{attribute addProperty BoxType "EL6201-0000-0017"}
{attribute addProperty Id "Slave_28A_DI0BIT10.125217Slave_28A_DI1BIT10.125218Slave_28A_DI2BIT10.125219Slave_28A_DI3BIT10.125220Slave_28B_DI0BIT10.125221Slave_28B_DI1BIT10.125222Slave_28B_DI2BIT10.125223Slave_28B_DI3BIT10.125224"}
{attribute addProperty CRC "1401413082"}
{attribute addProperty SizeInBites "8"}
{attribute addProperty SizeInBytes "1"}
TYPE Slave_28_Inputs_5387DDDA :
STRUCT
	{attribute addProperty Name "Slave_28A_DI0"}
	Slave_28A_DI0 : BIT;
	{attribute addProperty Name "Slave_28A_DI1"}
	Slave_28A_DI1 : BIT;
	{attribute addProperty Name "Slave_28A_DI2"}
	Slave_28A_DI2 : BIT;
	{attribute addProperty Name "Slave_28A_DI3"}
	Slave_28A_DI3 : BIT;
	{attribute addProperty Name "Slave_28B_DI0"}
	Slave_28B_DI0 : BIT;
	{attribute addProperty Name "Slave_28B_DI1"}
	Slave_28B_DI1 : BIT;
	{attribute addProperty Name "Slave_28B_DI2"}
	Slave_28B_DI2 : BIT;
	{attribute addProperty Name "Slave_28B_DI3"}
	Slave_28B_DI3 : BIT;
END_STRUCT
END_TYPE

(* stored: Version 1.2.0.0, ProductVersion 3.1.4024.9
   DUT Slave_28_Inputs_5387DDDA: Id {67f11f2e-e415-4174-86b5-c1cb6a5e60f1} *)
